// Mitsubishi GX Works2 project: 231004-002- exercicios   PLC: Q03UDV

// task Task_01 (event TRUE, interval 0, priority 31): POU_01
// task st_Prog2 (event TRUE, interval 0, priority 31): st_Prog2

PROGRAM POU_01
;
END_PROGRAM

FUNCTION f_soma
VAR_INPUT
  i_Valor1 : INT;
  i_Valor2 : INT;
END_VAR
f_soma := i_Valor1 + i_Valor2;
END_FUNCTION

PROGRAM st_Prog2
;
END_PROGRAM

FUNCTION f_Sub
VAR_INPUT
  i_Valor1 : INT;
  i_Valor2 : INT;
END_VAR
f_Sub := i_Valor1 - i_Valor2;
END_FUNCTION

FUNCTION f_mult
VAR_INPUT
  i_Valor1 : INT;
  i_Valor2 : INT;
END_VAR
f_mult := i_Valor1 * i_Valor2;
END_FUNCTION

FUNCTION f_div
VAR_INPUT
  i_Valor1 : INT;
  i_Valor2 : INT;
END_VAR
f_div := i_Valor1 / i_Valor2;
END_FUNCTION

FUNCTION_BLOCK operacoes
VAR_INPUT
  i_xValor1 : INT;
  i_xValor2 : INT;
END_VAR
VAR_OUTPUT
  o_ySoma : INT;
  o_ySub : INT;
  o_yMult : ARRAY [0..4] OF INT;
  o_yDiv : ARRAY [0..4] OF INT;
END_VAR

END_FUNCTION_BLOCK
